Staubli VAL3: OnF3.pgx

public program OnF3()
begin
end
